// TIA Portal V17 export
// export: Created 2022-05-07T16:38:49.0738123Z, ExportSetting WithDefaults, DisplayName Totally Integrated Automation Portal, DisplayVersion V17 Update 3, DisplayName TIA Portal Openness, DisplayVersion V17 Update 3, DisplayName TIA Portal Version Control Interface, DisplayVersion V17, DisplayName TIA Portal Test Suite Advanced, DisplayVersion V17 Update 1, DisplayName SINAMICS Startdrive Advanced, DisplayVersion V17 Update2, DisplayName SINAMICS Startdrive G130, G150, S120, S150, SINAMICS MV, S210, DisplayVersion V17 Update2, DisplayName SINAMICS Startdrive G110M, G120, G120C, G120D, G120P, G115D, DisplayVersion V17 Update2, DisplayName STEP 7 Professional, DisplayVersion V17 Update 3, DisplayName STEP 7 Safety, DisplayVersion V17, DisplayName WinCC UA Professional, DisplayVersion V17 Update 3
TYPE "UDTMotori"
// stored: IsFailsafeCompliant false
   STRUCT
      pos : Struct
         "1" : Real;
         "2" : Real;
         "3" : Real;
         "4" : Real;
         "5" : Real;
      END_STRUCT;
      vel : Struct
         "1" : Real;
         "2" : Real;
         "3" : Real;
         "4" : Real;
         "5" : Real;
      END_STRUCT;
      acc : Struct
         "1" : Real;
         "2" : Real;
         "3" : Real;
         "4" : Real;
         "5" : Real;
      END_STRUCT;
      dec : Struct
         "1" : Real;
         "2" : Real;
         "3" : Real;
         "4" : Real;
         "5" : Real;
      END_STRUCT;
      IN : Struct
         Exe_MC_Reset : Bool;   // comando di reset
         En_MC_Power : Bool;   // abilitazione asse
         Exe_MC_Home : Bool;   // comando di homing
         Sp_Offset_Homing : Real;   // offset azzeramento
         Exe_MC_Halt : Bool;   // comando HALT
         Exe_Jog_Fwd : Bool;   // comando jog +
         Exe_Jog_Bkw : Bool;   // comando jog -
         Sp_Jog_Velocity : Real;   // set velocità JOG
         Exe_MC_Velocity : Bool;   // comando velocità
         Sp_MC_Velocity : Real;   // set velocità Move Velocity
         Exe_MC_MoveRelative : Bool;   // comando posizione relativa
         Sp_MoveRel_Distance : Real;   // set distanza Move Relative
         Sp_MoveRel_Velocity : Real;   // set velocità Move Relative
         Exe_MC_MoveAbs : Bool;   // comando posizione assoluta
         Sp_MoveAbs_Position : Real;   // set posizione Move Absolute
         Sp_MoveAbs_Velocity : Real;   // set velocità Move Absolute
         Exe_MC_ChangeDyna : Bool;   // comando cambio dinamica
         Sp_RampUpTime : Real;   // set tempo di rampa acc [s]
         Sp_RampDnTime : Real;   // set tempo di rampa dec [s]
      END_STRUCT;
      OUT : Struct
         Output_MC_Reset_Done : Bool;   // asse resettato
         Output_MC_AxisEnabled : Bool;   // asse abilitato
         Output_MC_AxisHomed : Bool;   // asse homed (referenziato)
         Output_MC_Halt_Done : Bool;   // asse in halt
         Output_MC_JogInVelocity : Bool;   // vel raggiunta
         Output_MC_MoveInVelocity : Bool;   // vel raggiunta
         Output_MC_MoveRel_Done : Bool;   // move realtive eseguito
         Output_MC_MoveAbs_Done : Bool;   // move absolute eseguito
         Output_MC_MoveAbs_Busy : Bool;   // move absolute in corso
         Output_MC_At_Standstill : Bool;   // asse fermo
         Output_MC_Error : Bool;   // asse in errore (or di vari bool)
         Output_ActVelocity : Real;   // velocity attuale (asse)
         Output_ActPos : Real;   // posizione attuale
      END_STRUCT;
   END_STRUCT;
END_TYPE
